Fanuc KAREL source: RGET_REG.kl

PROGRAM T
%NOLOCKGROUP
VAR
 v0 : STRING[40]
 v1 : BOOLEAN
 v2 : INTEGER
 v3 : INTEGER
 v4 : REAL
 v5 : INTEGER
BEGIN
 RGET_REG(v0, v1, v2, v3, v4, v5)
END T
